FUNCTION CheckDivReal : REAL
VAR_INPUT
	divisor		 		: REAL;
END_VAR
VAR
END_VAR

IF divisor = 0 THEN
	CheckRealZeroDiv_ErrCnt := CheckRealZeroDiv_ErrCnt + 1;
	CheckDivReal := 1;
ELSE
	CheckDivReal := divisor;
END_IF

END_FUNCTION

(* stored: Version 1.1.0.1, ProductVersion 3.1.4024.9
   POU CheckDivReal: Id {1054d4d6-15f8-4e7d-bd8b-11b64a27754c}, SpecialFunc CheckDivReal32 *)
